(* IEC 61131-3 sources: Std_PalletMover/Class/HwI_BasicLift, 1 file *)

(* ---- HwI_BasicLift.st ---- *)
(*!
<Class
	Name               = "HwI_BasicLift"
	Revision           = "0.0"
	RealtimeTask       = "false"
	CyclicTask         = "false"
	BackgroundTask     = "false"
	Sigmatek           = "false"
	OSInterface        = "false"
	HighPriority       = "false"
	Automatic          = "false"
	UpdateMode         = "Prescan"
	SharedCommandTable = "true"
	Objectsize         = "(570,120)">
	<Channels>
		<Server Name="ClassSvr" Visualized="false" Initialize="false" WriteProtected="true" Retentive="false"/>
		<Client Name="ActuatorValveDown" Required="true" Internal="false"/>
		<Client Name="ActuatorValveUp" Required="true" Internal="false"/>
		<Client Name="Ain_AnalogPosition" Required="true" Internal="false"/>
		<Client Name="SensorMaxHeight" Required="true" Internal="false"/>
		<Client Name="SensorMinHeight" Required="true" Internal="false"/>
		<Client Name="Speed" Required="true" Internal="false"/>
	</Channels>
</Class>
*)
HwI_BasicLift : CLASS
  //Servers:
	ClassSvr 	: SvrChCmd_DINT;
  //Clients:
	Ain_AnalogPosition 	: CltCh_DINT;
	SensorMaxHeight 	: CltCh_DINT;
	SensorMinHeight 	: CltCh_DINT;
	ActuatorValveUp 	: CltCh_DINT;
	ActuatorValveDown 	: CltCh_DINT;
	Speed 	: CltCh_DINT;
  //Variables:
  //Functions:
  //Tables:
	FUNCTION @STD
		VAR_OUTPUT
			ret_code	: CONFSTATES;
		END_VAR;
	FUNCTION GLOBAL TAB @CT_;
END_CLASS;
